(* Logix 5000 project; controller TBEN_Lx_8IOL_AOI_V0_1 vendor 1 type 14 code 176 rev 32.11; software revision 32.00; part 9 of 11 *)
(* tags used below, declared in another part *)
   IOLReadActive : BOOL;
   IOLWriteActive : BOOL;
   IOL_READ_Request : BOOL;
   IOL_WRITE_Request : BOOL;
(* TBEN_Lx_8IOL_AOI, continued *)

ROUTINE Prescan   (* ladder *)
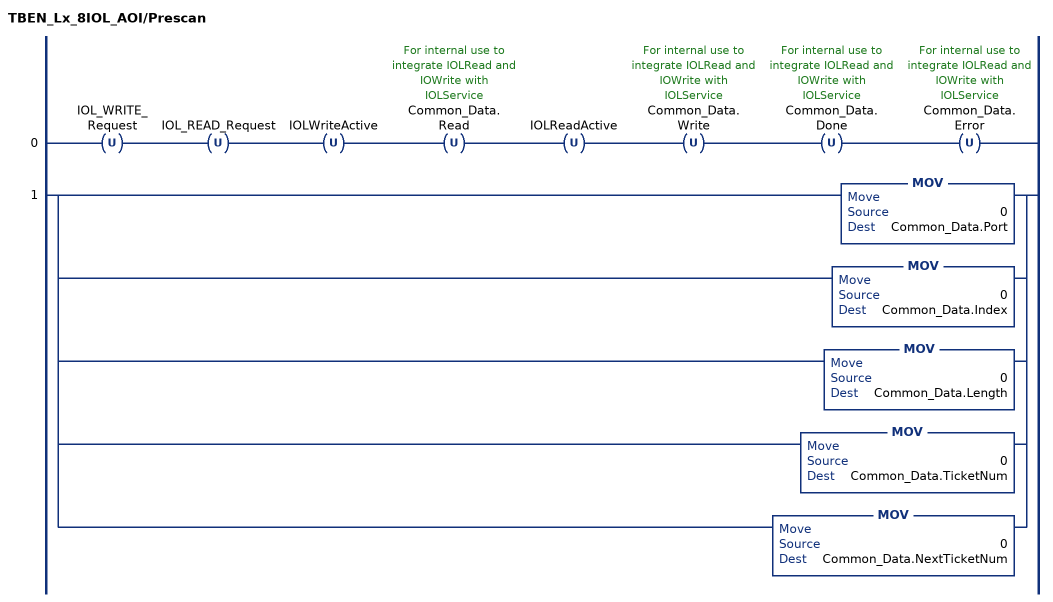
   0: OTU(IOL_WRITE_Request)OTU(IOL_READ_Request)OTU(IOLWriteActive)OTU(Common_Data.Read)OTU(IOLReadActive)OTU(Common_Data.Write)OTU(Common_Data.Done)OTU(Common_Data.Error);
   1: [MOV(0,Common_Data.Port) ,MOV(0,Common_Data.Index) ,MOV(0,Common_Data.Length) ,MOV(0,Common_Data.TicketNum) ,MOV(0,Common_Data.NextTicketNum) ];
END_ROUTINE
END_ADD_ON_INSTRUCTION

ADD_ON_INSTRUCTION Universal_Device_Info   (* revision 1.0, ExecutePrescan *)
VAR_INPUT
   Port : INT; {required}
END_VAR
VAR_IN_OUT
   Common_Data : Turck_IOLink_Common_Data; {required}
END_VAR
VAR_INPUT
   Write_Application_Specific_Tag : BOOL;
END_VAR
VAR_IN_OUT
   Universal_IOLink_Info : Universal_IOLink_Info; {required}
END_VAR
VAR
   StartupDone : BOOL; {access None}
   Done : DINT; {access None}
   Error : DINT; {access None}
   Active : DINT; {access None}
   Pending : DINT; {access None}
   Pending_or_Active : DINT; {access None}
   StartupCount : DINT; {access None}
   MyTicketNum : DINT[32]; {access None}
   Read_ONS : DINT; {access None}
   ReadRequest : DINT; {access None}
   Read : DINT; {access None}
   DoneCount : DINT; {access None}
   Status : DINT; {access None}
   ErrorCount : DINT; {access None}
   Prev_Vendor_ID : INT; {access None}
   Update_Data : BOOL; {access None}
   Reset : BOOL; {access None}
   Write_ONS : DINT; {access None}
   WriteRequest : DINT; {access None}
END_VAR

ROUTINE Logic   (* ladder *)
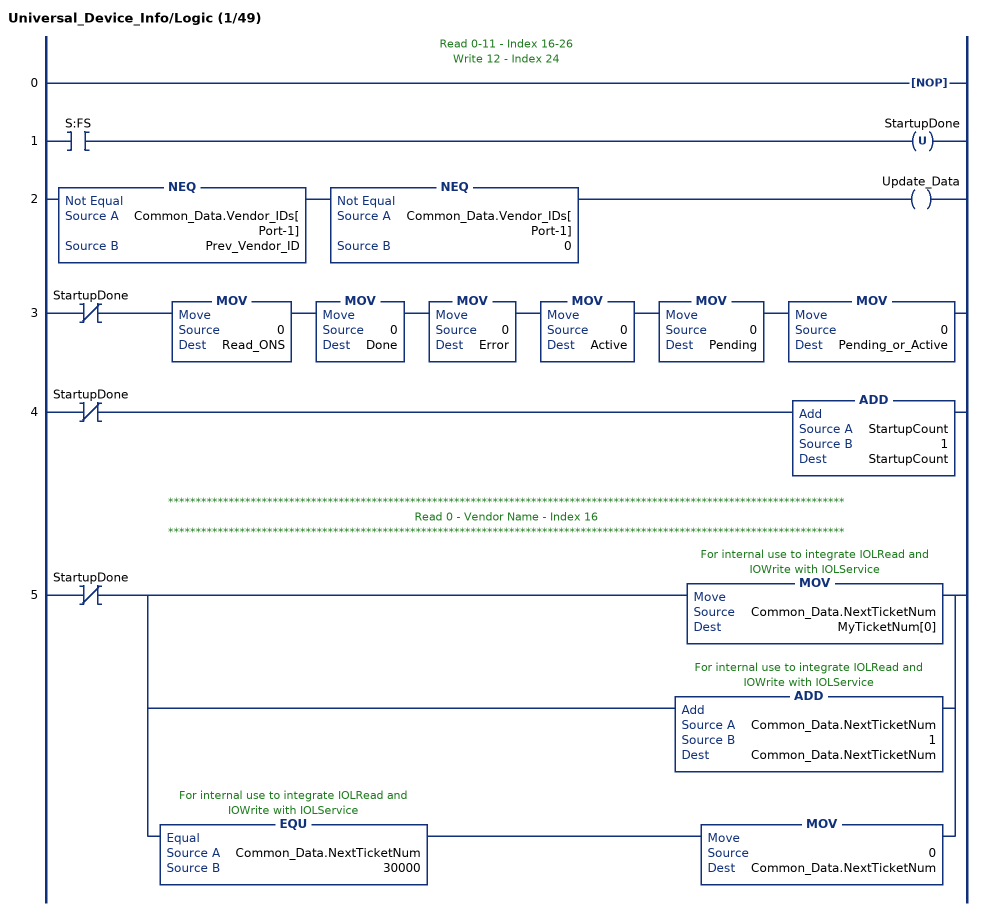
   // Read 0-11 - Index 16-26
   // Write 12 - Index 24
   0: NOP();
   1: XIC(S:FS)OTU(StartupDone);
   2: NEQ(Common_Data.Vendor_IDs[Port-1],Prev_Vendor_ID)NEQ(Common_Data.Vendor_IDs[Port-1],0)OTE(Update_Data);
   3: XIO(StartupDone)MOV(0,Read_ONS)MOV(0,Done)MOV(0,Error)MOV(0,Active)MOV(0,Pending)MOV(0,Pending_or_Active);
   4: XIO(StartupDone)ADD(StartupCount,1,StartupCount);
   // ***************************************************************************************************************************
   // Read 0 - Vendor Name - Index 16
   // ***************************************************************************************************************************
   5: XIO(StartupDone)[MOV(Common_Data.NextTicketNum,MyTicketNum[0]) ,ADD(Common_Data.NextTicketNum,1,Common_Data.NextTicketNum) ,EQU(Common_Data.NextTicketNum,30000) MOV(0,Common_Data.NextTicketNum) ];
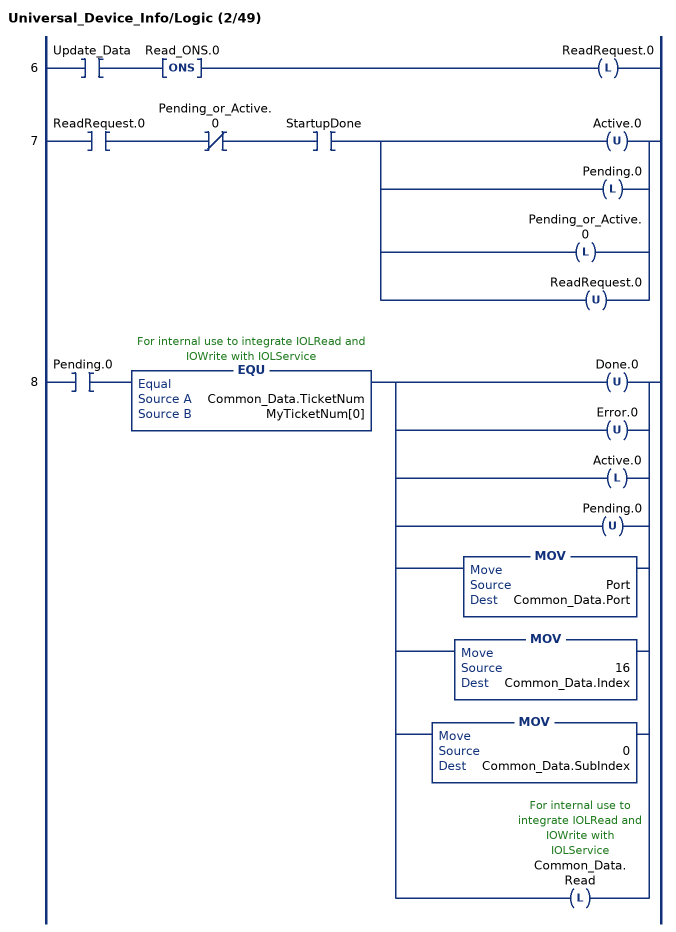
   6: XIC(Update_Data)ONS(Read_ONS.0)OTL(ReadRequest.0);
   7: XIC(ReadRequest.0)XIO(Pending_or_Active.0)XIC(StartupDone)[OTU(Active.0) ,OTL(Pending.0) ,OTL(Pending_or_Active.0) ,OTU(ReadRequest.0) ];
   8: XIC(Pending.0)EQU(Common_Data.TicketNum,MyTicketNum[0])[OTU(Done.0) ,OTU(Error.0) ,OTL(Active.0) ,OTU(Pending.0) ,MOV(Port,Common_Data.Port) ,MOV(16,Common_Data.Index) ,MOV(0,Common_Data.SubIndex) ,OTL(Common_Data.Read) ];
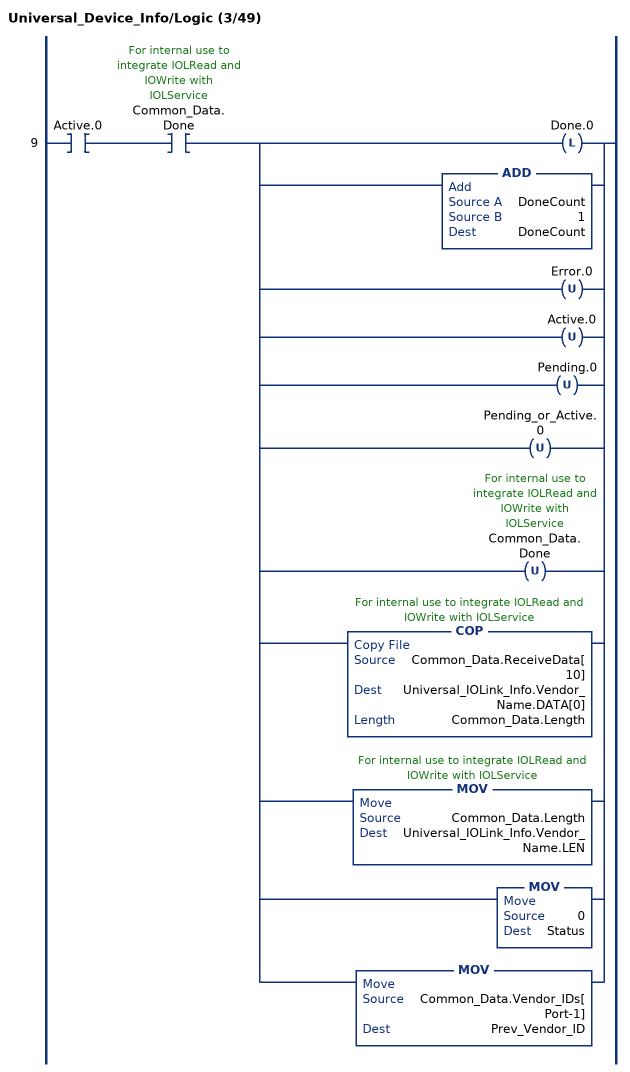
   9: XIC(Active.0)XIC(Common_Data.Done)[OTL(Done.0) ,ADD(DoneCount,1,DoneCount) ,OTU(Error.0) ,OTU(Active.0) ,OTU(Pending.0) ,OTU(Pending_or_Active.0) ,OTU(Common_Data.Done) ,COP(Common_Data.ReceiveData[10],Universal_IOLink_Info.Vendor_Name.DATA[0],Common_Data.Length) ,MOV(Common_Data.Length,Universal_IOLink_Info.Vendor_Name.LEN) ,MOV(0,Status) ,MOV(Common_Data.Vendor_IDs[Port-1],Prev_Vendor_ID) ];
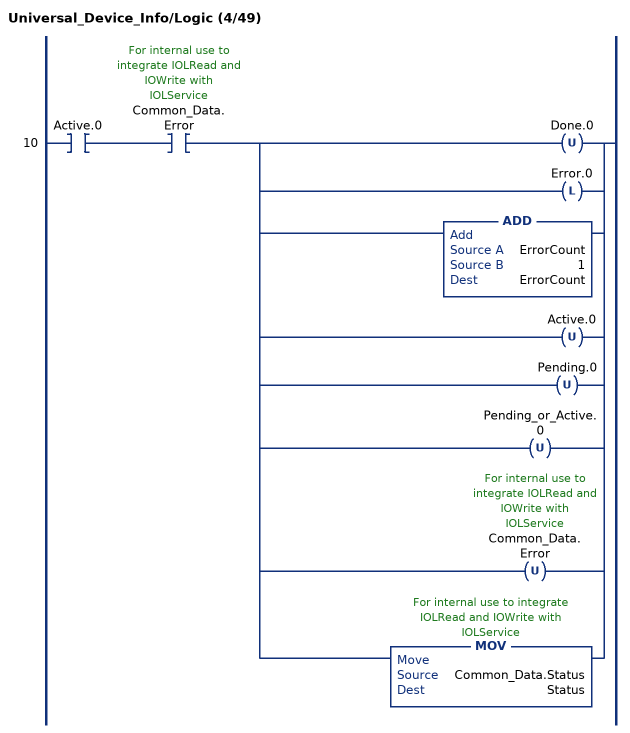
   10: XIC(Active.0)XIC(Common_Data.Error)[OTU(Done.0) ,OTL(Error.0) ,ADD(ErrorCount,1,ErrorCount) ,OTU(Active.0) ,OTU(Pending.0) ,OTU(Pending_or_Active.0) ,OTU(Common_Data.Error) ,MOV(Common_Data.Status,Status) ];
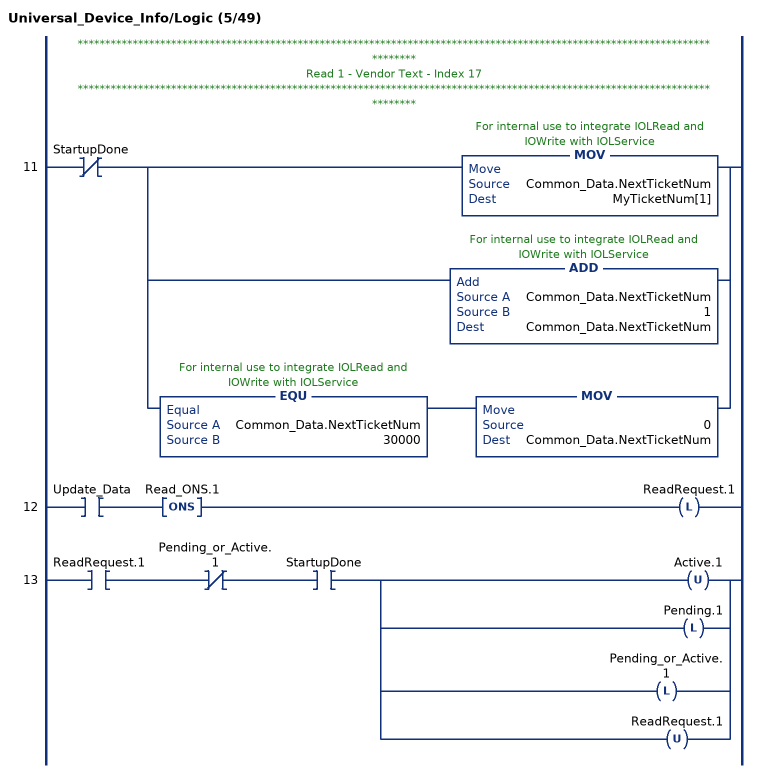
   // ***************************************************************************************************************************
   // Read 1 - Vendor Text - Index 17
   // ***************************************************************************************************************************
   11: XIO(StartupDone)[MOV(Common_Data.NextTicketNum,MyTicketNum[1]) ,ADD(Common_Data.NextTicketNum,1,Common_Data.NextTicketNum) ,EQU(Common_Data.NextTicketNum,30000) MOV(0,Common_Data.NextTicketNum) ];
   12: XIC(Update_Data)ONS(Read_ONS.1)OTL(ReadRequest.1);
   13: XIC(ReadRequest.1)XIO(Pending_or_Active.1)XIC(StartupDone)[OTU(Active.1) ,OTL(Pending.1) ,OTL(Pending_or_Active.1) ,OTU(ReadRequest.1) ];
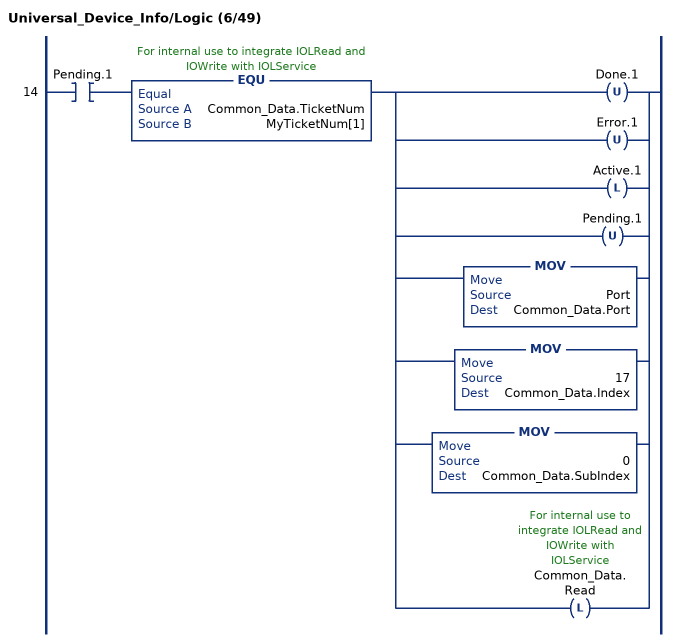
   14: XIC(Pending.1)EQU(Common_Data.TicketNum,MyTicketNum[1])[OTU(Done.1) ,OTU(Error.1) ,OTL(Active.1) ,OTU(Pending.1) ,MOV(Port,Common_Data.Port) ,MOV(17,Common_Data.Index) ,MOV(0,Common_Data.SubIndex) ,OTL(Common_Data.Read) ];
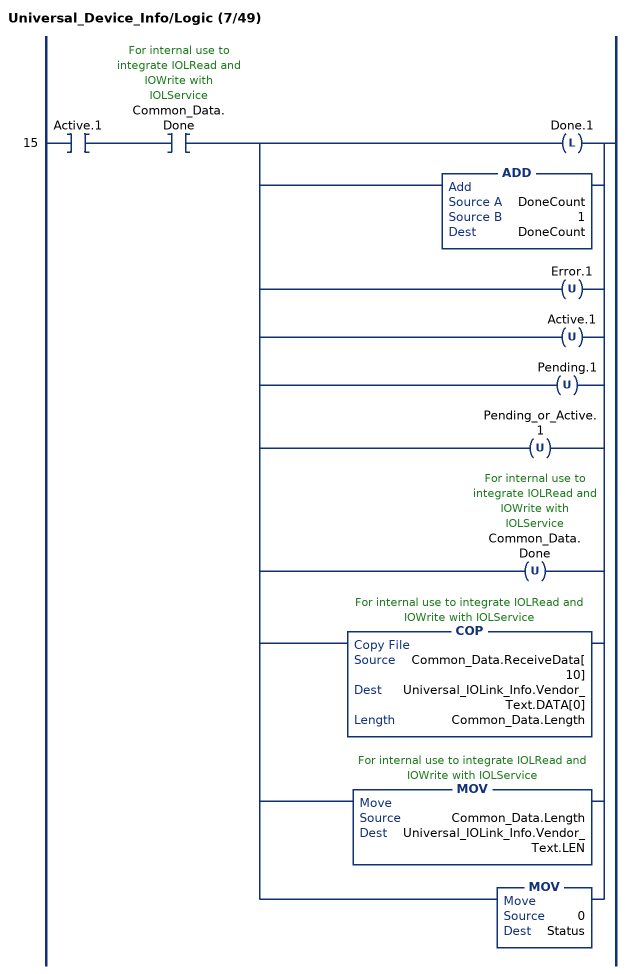
   15: XIC(Active.1)XIC(Common_Data.Done)[OTL(Done.1) ,ADD(DoneCount,1,DoneCount) ,OTU(Error.1) ,OTU(Active.1) ,OTU(Pending.1) ,OTU(Pending_or_Active.1) ,OTU(Common_Data.Done) ,COP(Common_Data.ReceiveData[10],Universal_IOLink_Info.Vendor_Text.DATA[0],Common_Data.Length) ,MOV(Common_Data.Length,Universal_IOLink_Info.Vendor_Text.LEN) ,MOV(0,Status) ];
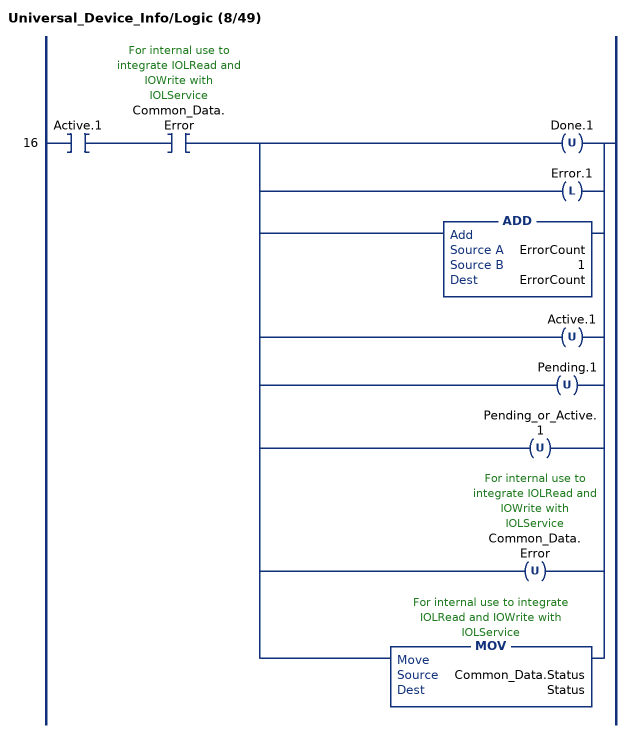
   16: XIC(Active.1)XIC(Common_Data.Error)[OTU(Done.1) ,OTL(Error.1) ,ADD(ErrorCount,1,ErrorCount) ,OTU(Active.1) ,OTU(Pending.1) ,OTU(Pending_or_Active.1) ,OTU(Common_Data.Error) ,MOV(Common_Data.Status,Status) ];
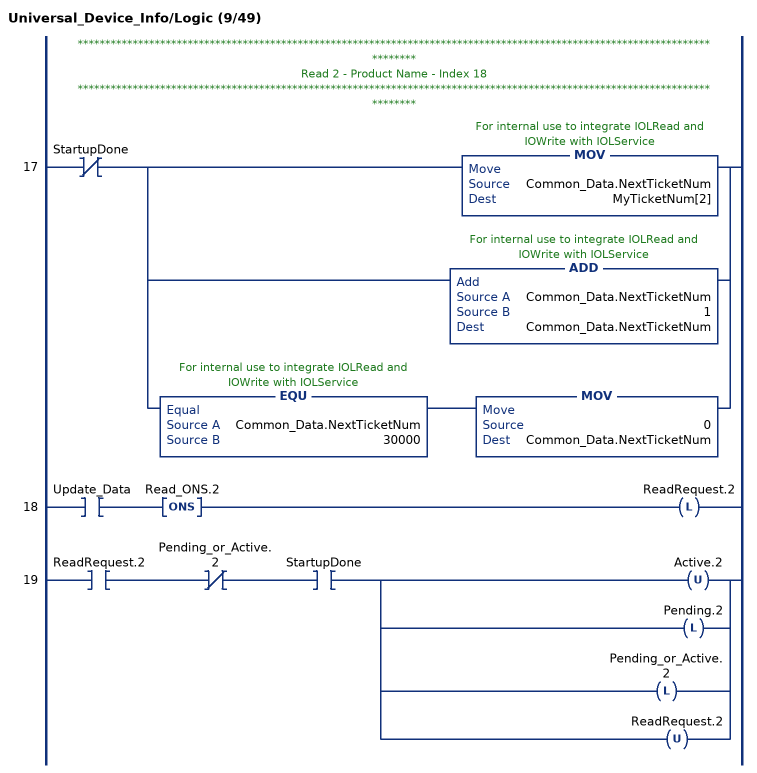
   // ***************************************************************************************************************************
   // Read 2 - Product Name - Index 18
   // ***************************************************************************************************************************
   17: XIO(StartupDone)[MOV(Common_Data.NextTicketNum,MyTicketNum[2]) ,ADD(Common_Data.NextTicketNum,1,Common_Data.NextTicketNum) ,EQU(Common_Data.NextTicketNum,30000) MOV(0,Common_Data.NextTicketNum) ];
   18: XIC(Update_Data)ONS(Read_ONS.2)OTL(ReadRequest.2);
   19: XIC(ReadRequest.2)XIO(Pending_or_Active.2)XIC(StartupDone)[OTU(Active.2) ,OTL(Pending.2) ,OTL(Pending_or_Active.2) ,OTU(ReadRequest.2) ];
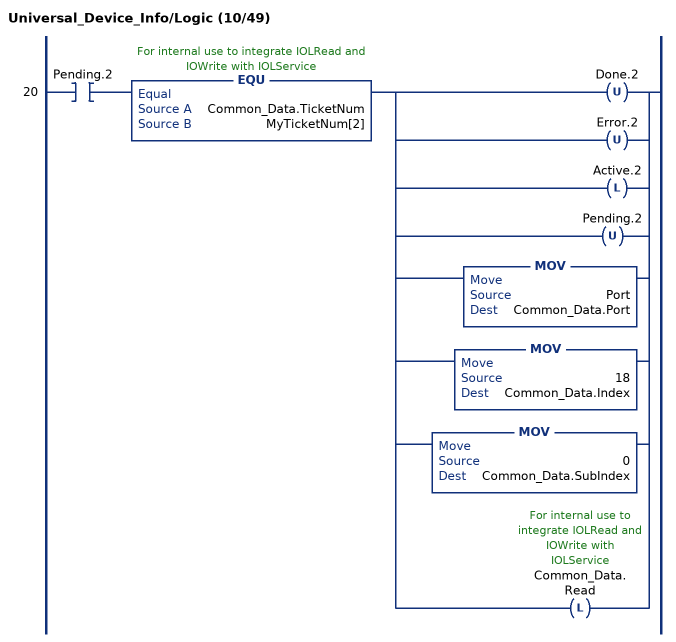
   20: XIC(Pending.2)EQU(Common_Data.TicketNum,MyTicketNum[2])[OTU(Done.2) ,OTU(Error.2) ,OTL(Active.2) ,OTU(Pending.2) ,MOV(Port,Common_Data.Port) ,MOV(18,Common_Data.Index) ,MOV(0,Common_Data.SubIndex) ,OTL(Common_Data.Read) ];
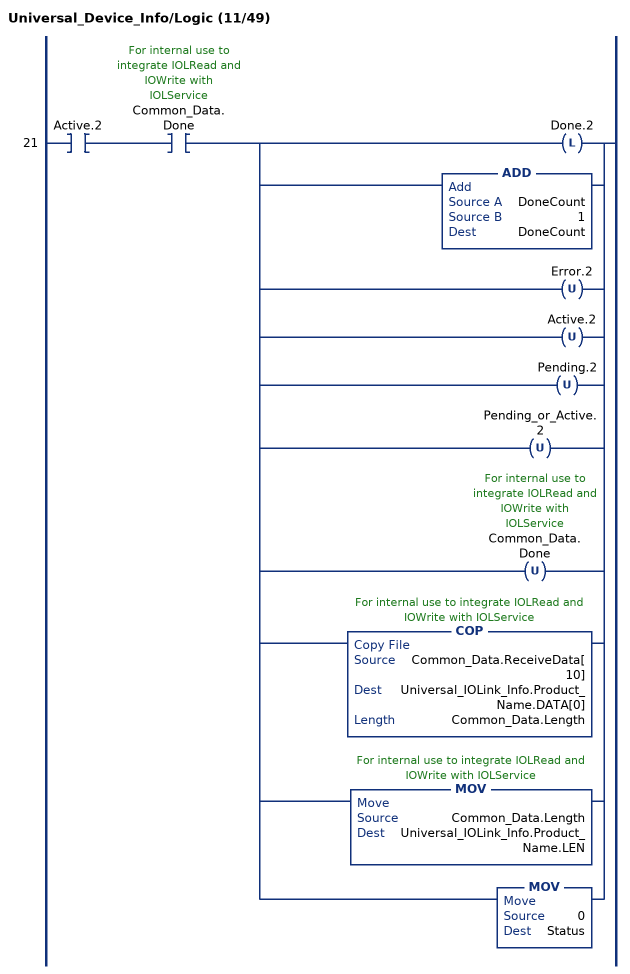
   21: XIC(Active.2)XIC(Common_Data.Done)[OTL(Done.2) ,ADD(DoneCount,1,DoneCount) ,OTU(Error.2) ,OTU(Active.2) ,OTU(Pending.2) ,OTU(Pending_or_Active.2) ,OTU(Common_Data.Done) ,COP(Common_Data.ReceiveData[10],Universal_IOLink_Info.Product_Name.DATA[0],Common_Data.Length) ,MOV(Common_Data.Length,Universal_IOLink_Info.Product_Name.LEN) ,MOV(0,Status) ];
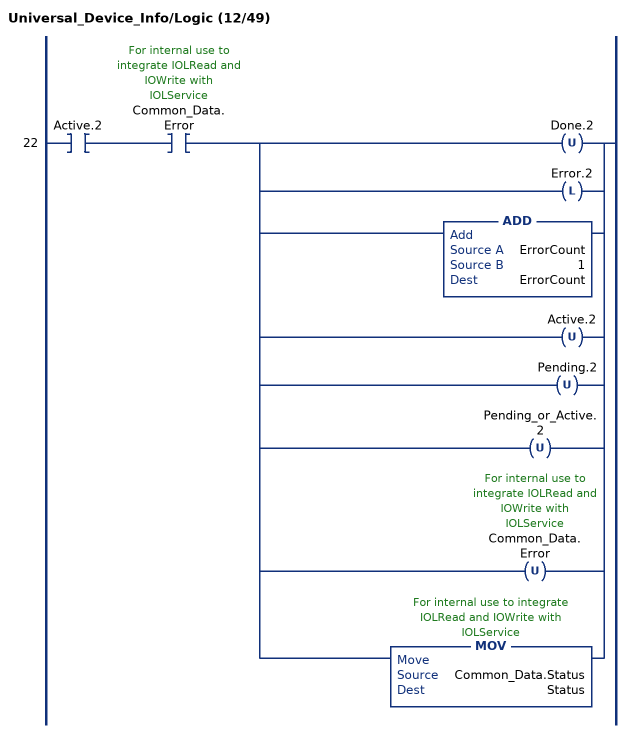
   22: XIC(Active.2)XIC(Common_Data.Error)[OTU(Done.2) ,OTL(Error.2) ,ADD(ErrorCount,1,ErrorCount) ,OTU(Active.2) ,OTU(Pending.2) ,OTU(Pending_or_Active.2) ,OTU(Common_Data.Error) ,MOV(Common_Data.Status,Status) ];
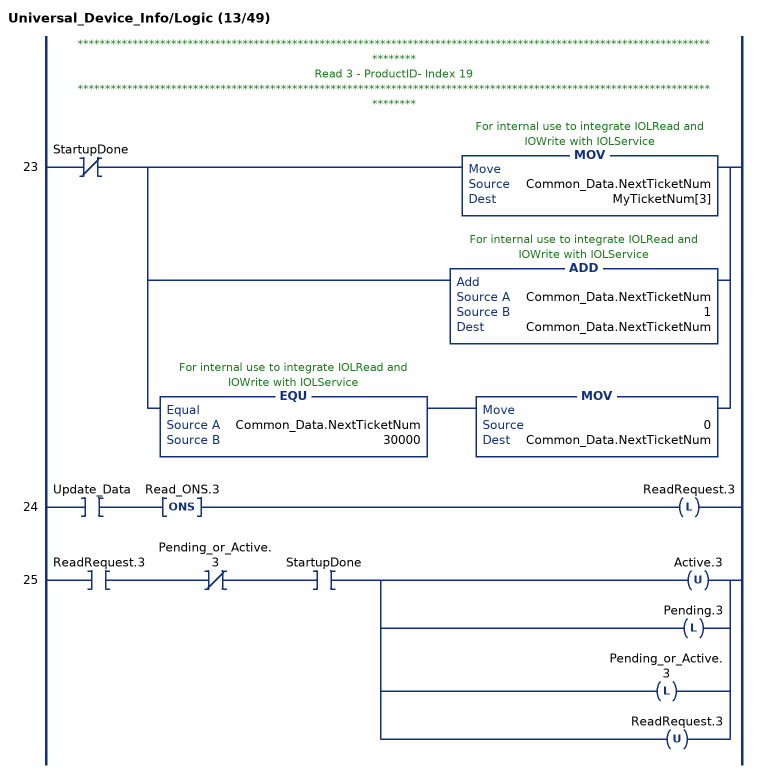
   // ***************************************************************************************************************************
   // Read 3 - ProductID- Index 19
   // ***************************************************************************************************************************
   23: XIO(StartupDone)[MOV(Common_Data.NextTicketNum,MyTicketNum[3]) ,ADD(Common_Data.NextTicketNum,1,Common_Data.NextTicketNum) ,EQU(Common_Data.NextTicketNum,30000) MOV(0,Common_Data.NextTicketNum) ];
   24: XIC(Update_Data)ONS(Read_ONS.3)OTL(ReadRequest.3);
   25: XIC(ReadRequest.3)XIO(Pending_or_Active.3)XIC(StartupDone)[OTU(Active.3) ,OTL(Pending.3) ,OTL(Pending_or_Active.3) ,OTU(ReadRequest.3) ];
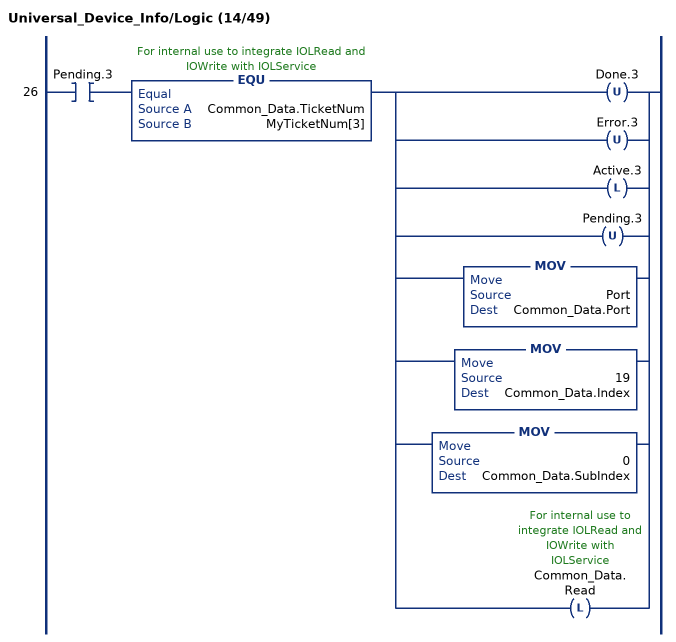
   26: XIC(Pending.3)EQU(Common_Data.TicketNum,MyTicketNum[3])[OTU(Done.3) ,OTU(Error.3) ,OTL(Active.3) ,OTU(Pending.3) ,MOV(Port,Common_Data.Port) ,MOV(19,Common_Data.Index) ,MOV(0,Common_Data.SubIndex) ,OTL(Common_Data.Read) ];
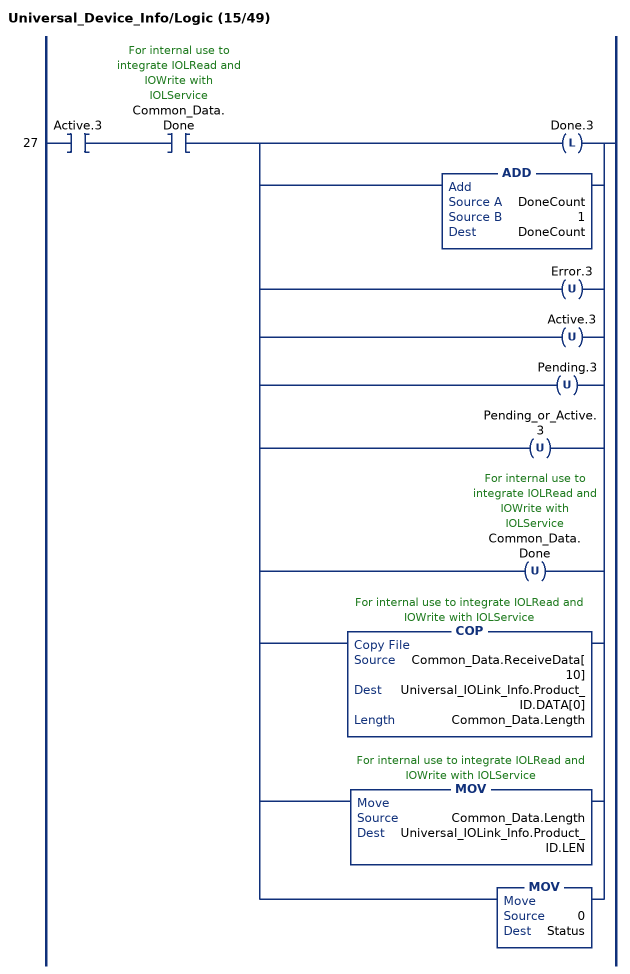
   27: XIC(Active.3)XIC(Common_Data.Done)[OTL(Done.3) ,ADD(DoneCount,1,DoneCount) ,OTU(Error.3) ,OTU(Active.3) ,OTU(Pending.3) ,OTU(Pending_or_Active.3) ,OTU(Common_Data.Done) ,COP(Common_Data.ReceiveData[10],Universal_IOLink_Info.Product_ID.DATA[0],Common_Data.Length) ,MOV(Common_Data.Length,Universal_IOLink_Info.Product_ID.LEN) ,MOV(0,Status) ];
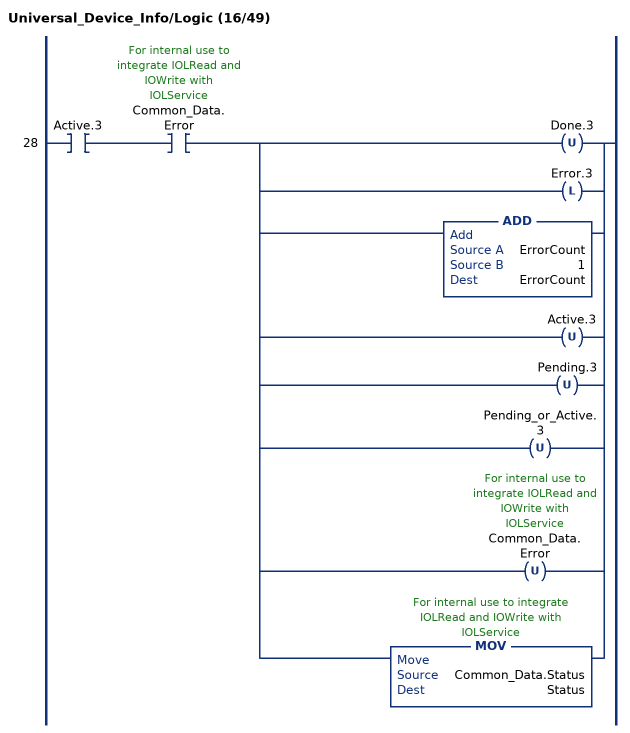
   28: XIC(Active.3)XIC(Common_Data.Error)[OTU(Done.3) ,OTL(Error.3) ,ADD(ErrorCount,1,ErrorCount) ,OTU(Active.3) ,OTU(Pending.3) ,OTU(Pending_or_Active.3) ,OTU(Common_Data.Error) ,MOV(Common_Data.Status,Status) ];
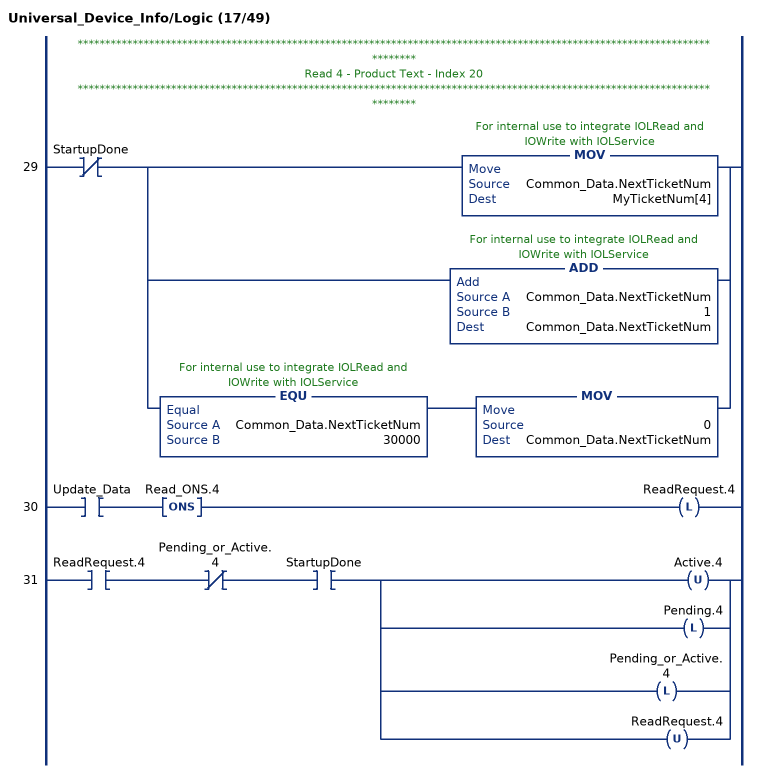
   // ***************************************************************************************************************************
   // Read 4 - Product Text - Index 20
   // ***************************************************************************************************************************
   29: XIO(StartupDone)[MOV(Common_Data.NextTicketNum,MyTicketNum[4]) ,ADD(Common_Data.NextTicketNum,1,Common_Data.NextTicketNum) ,EQU(Common_Data.NextTicketNum,30000) MOV(0,Common_Data.NextTicketNum) ];
   30: XIC(Update_Data)ONS(Read_ONS.4)OTL(ReadRequest.4);
   31: XIC(ReadRequest.4)XIO(Pending_or_Active.4)XIC(StartupDone)[OTU(Active.4) ,OTL(Pending.4) ,OTL(Pending_or_Active.4) ,OTU(ReadRequest.4) ];
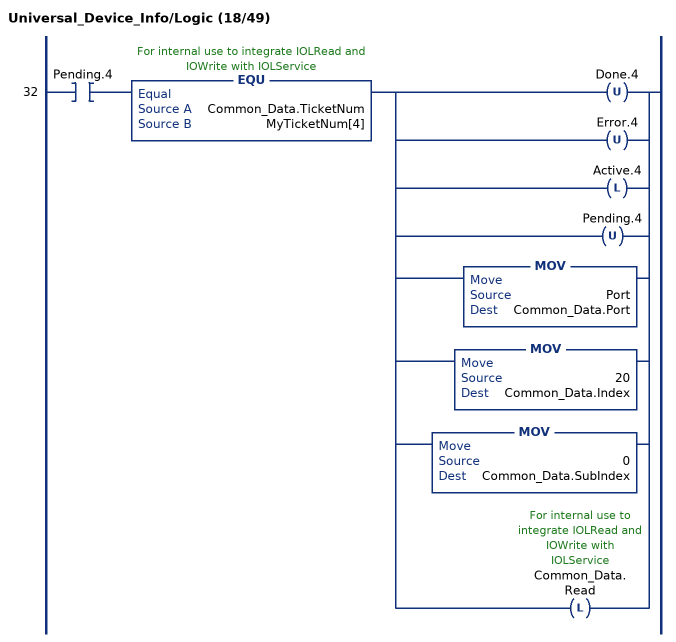
   32: XIC(Pending.4)EQU(Common_Data.TicketNum,MyTicketNum[4])[OTU(Done.4) ,OTU(Error.4) ,OTL(Active.4) ,OTU(Pending.4) ,MOV(Port,Common_Data.Port) ,MOV(20,Common_Data.Index) ,MOV(0,Common_Data.SubIndex) ,OTL(Common_Data.Read) ];
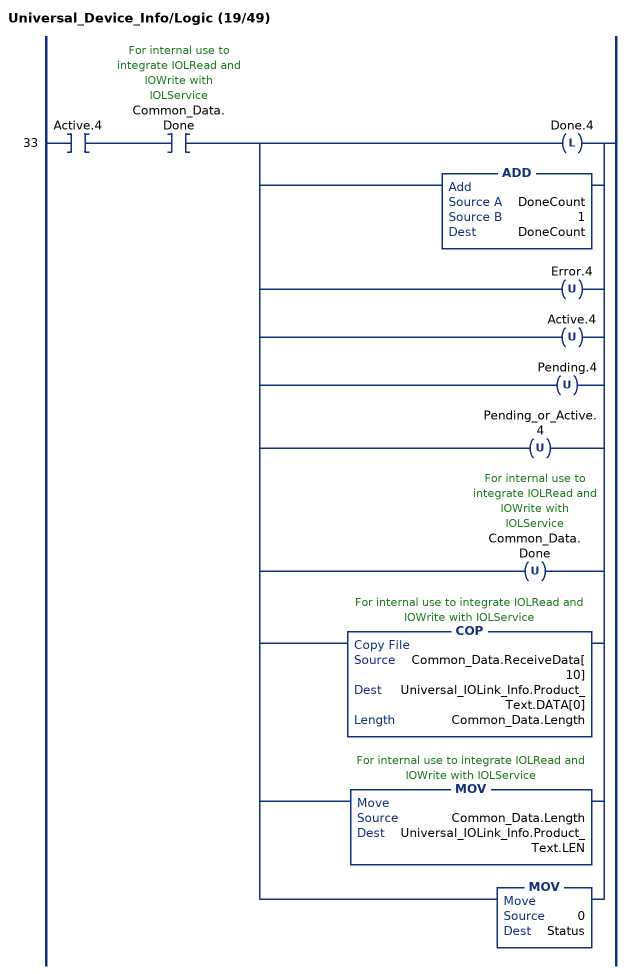
   33: XIC(Active.4)XIC(Common_Data.Done)[OTL(Done.4) ,ADD(DoneCount,1,DoneCount) ,OTU(Error.4) ,OTU(Active.4) ,OTU(Pending.4) ,OTU(Pending_or_Active.4) ,OTU(Common_Data.Done) ,COP(Common_Data.ReceiveData[10],Universal_IOLink_Info.Product_Text.DATA[0],Common_Data.Length) ,MOV(Common_Data.Length,Universal_IOLink_Info.Product_Text.LEN) ,MOV(0,Status) ];
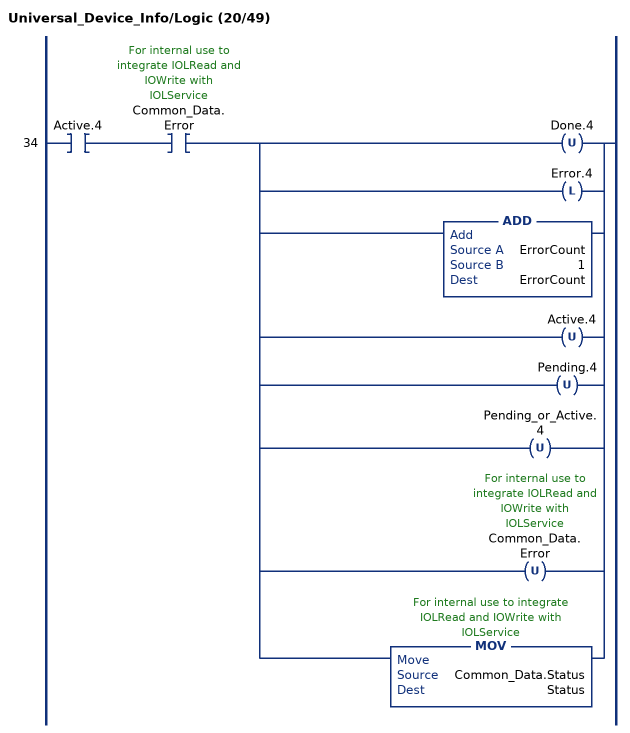
   34: XIC(Active.4)XIC(Common_Data.Error)[OTU(Done.4) ,OTL(Error.4) ,ADD(ErrorCount,1,ErrorCount) ,OTU(Active.4) ,OTU(Pending.4) ,OTU(Pending_or_Active.4) ,OTU(Common_Data.Error) ,MOV(Common_Data.Status,Status) ];
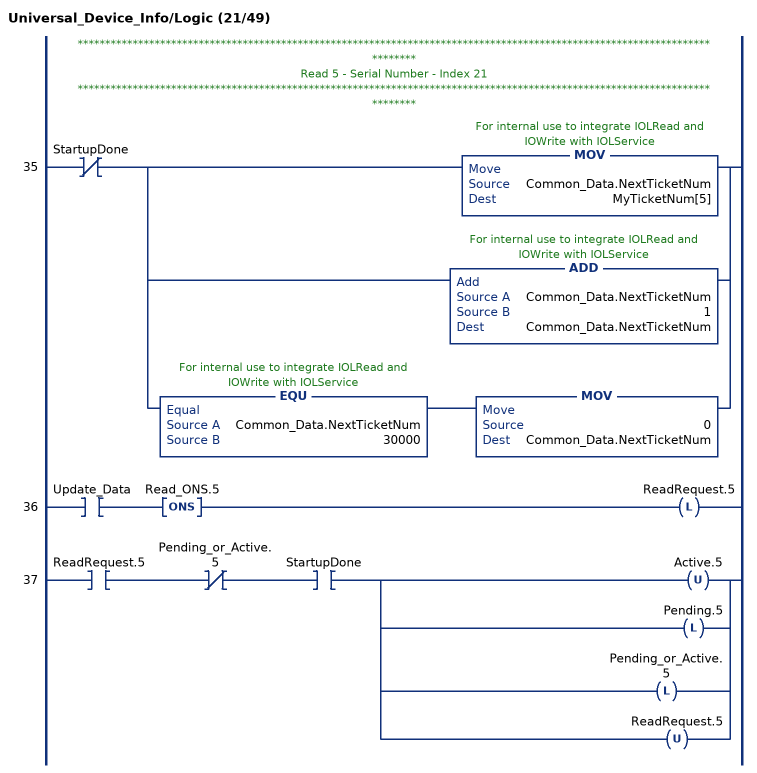
   // ***************************************************************************************************************************
   // Read 5 - Serial Number - Index 21
   // ***************************************************************************************************************************
   35: XIO(StartupDone)[MOV(Common_Data.NextTicketNum,MyTicketNum[5]) ,ADD(Common_Data.NextTicketNum,1,Common_Data.NextTicketNum) ,EQU(Common_Data.NextTicketNum,30000) MOV(0,Common_Data.NextTicketNum) ];
   36: XIC(Update_Data)ONS(Read_ONS.5)OTL(ReadRequest.5);
   37: XIC(ReadRequest.5)XIO(Pending_or_Active.5)XIC(StartupDone)[OTU(Active.5) ,OTL(Pending.5) ,OTL(Pending_or_Active.5) ,OTU(ReadRequest.5) ];
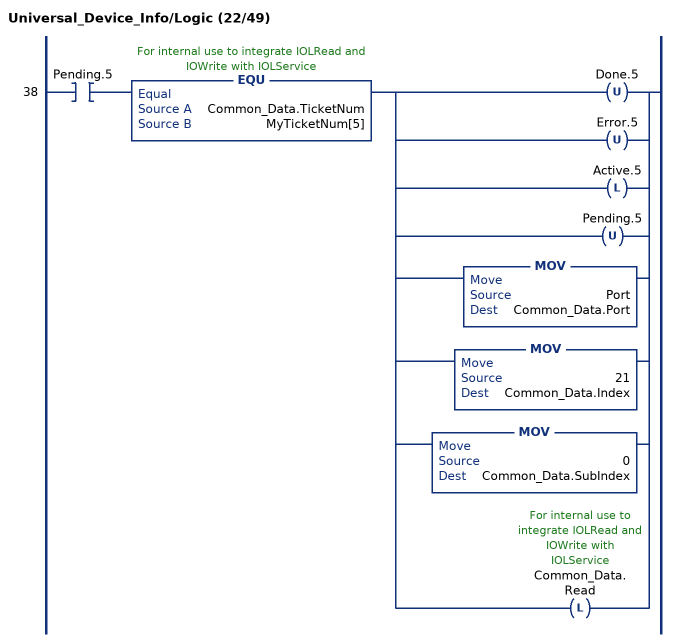
   38: XIC(Pending.5)EQU(Common_Data.TicketNum,MyTicketNum[5])[OTU(Done.5) ,OTU(Error.5) ,OTL(Active.5) ,OTU(Pending.5) ,MOV(Port,Common_Data.Port) ,MOV(21,Common_Data.Index) ,MOV(0,Common_Data.SubIndex) ,OTL(Common_Data.Read) ];
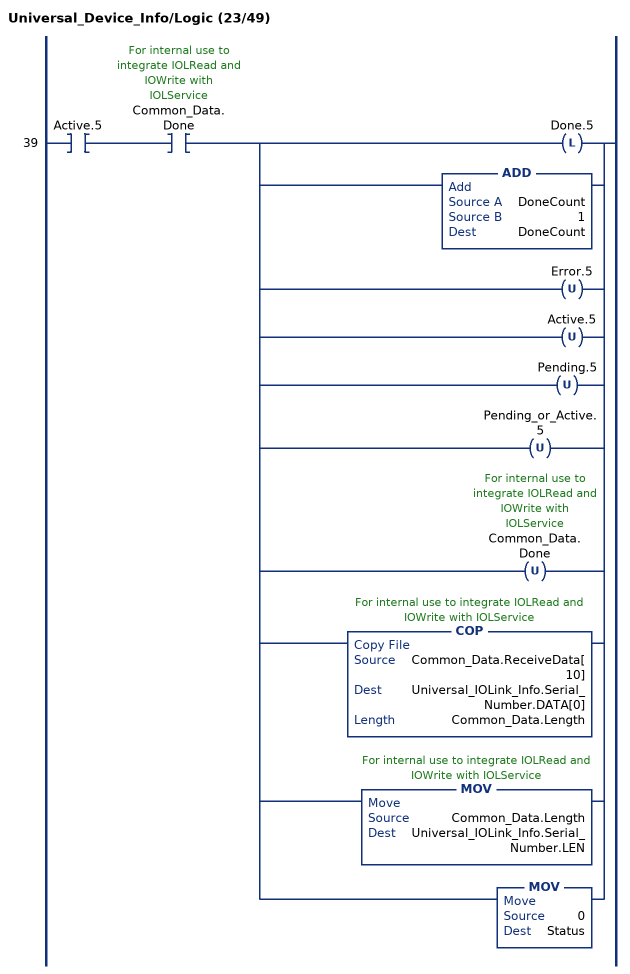
   39: XIC(Active.5)XIC(Common_Data.Done)[OTL(Done.5) ,ADD(DoneCount,1,DoneCount) ,OTU(Error.5) ,OTU(Active.5) ,OTU(Pending.5) ,OTU(Pending_or_Active.5) ,OTU(Common_Data.Done) ,COP(Common_Data.ReceiveData[10],Universal_IOLink_Info.Serial_Number.DATA[0],Common_Data.Length) ,MOV(Common_Data.Length,Universal_IOLink_Info.Serial_Number.LEN) ,MOV(0,Status) ];
